TYPE ST_TransportDataRequest :
(**************************************************************************************
 * 	Application		:	BoxControl Framework
 *	Revision		:	$Revision: 404529 $
 *	Revision date	:	$Date: 2018-04-23 08:21:38 +0200 (Mo., 23 Apr 2018) $
 *	Last changed by	:	$Author: b7bolm $
 *	URL				:	$URL: http://almscdc.swisslog.com/repo/SWPD/Development/BoxControlFramework/20_Release/trunk/01_Software/BCF/BCF/JumpStart/20_Product/10_App/12_E_Functions/10_Lib/10_Conv/10_Functions/01_DUTs/ST_TransportDataRequest.TcDUT $
 *
 *	Purpose			:	Transport control inputs
 *
 * ------------------------------------------------------------------------------------
 *	Copyright Swisslog [IP AG], Switzerland. All rights reserved.
 * 
 * ------------------------------------------------------------------------------------
 *	
 * 	Revision History: 
 *
 * 	VERSION			DATE			INITIALS			DESCRIPTION
 *	0.1				01.01.2001		swl					Example
 *
 **************************************************************************************)	
STRUCT
	RequestPrevTransportData : BOOL; // Request previous transport data
	RequestNextTransportData : BOOL; // Request next transport data
	DeletePrevTransportData	 : BOOL; // Delete previous transport data
	DeleteNextTransportData  : BOOL; // Delete next transport data
END_STRUCT
END_TYPE

(* stored: Version 1.1.0.1, ProductVersion 3.1.4022.12
   DUT ST_TransportDataRequest: Id {317aba52-5985-43c9-8891-64ce3d884ec5} *)
